// TwinCAT 3 PLC project Test_StopWatch_Level
// ProgramVersion: 3.1.4023.0
// libraries:
//   library_StopWatch_Level, * (Automatizaciones Adegar)
//   Tc2_Standard, * (Beckhoff Automation GmbH)
//   Tc2_System, * (Beckhoff Automation GmbH)
//   Tc3_Module, * (Beckhoff Automation GmbH)
// project tree:
//   / PlcTask.TcTTO
//   POUs/ MAIN.TcPOU
// (motion and I/O tree: see PLC project stopwatch_level)
// real-time tasks:
//   TASK PlcTask: cycle T#10ms, priority 20, ADS port 350

CONFIGURATION Test_StopWatch_Level
    RESOURCE PLC ON TwinCAT3
        TASK PlcTask(INTERVAL := T#10ms, PRIORITY := 20);
        PROGRAM MAIN WITH PlcTask : MAIN;
    END_RESOURCE
END_CONFIGURATION

// ---- POUs/MAIN.TcPOU
PROGRAM MAIN
VAR
	Stopwatch1 : FB_StopWatch_Level;
END_VAR

Stopwatch1(bSTART:= , bRESET:= , Elapsed_Time=> );

END_PROGRAM
